Staubli VAL3: gripper.pgx

public program gripper(num nOpen (dimensions=1))
begin
  //nOpen = 0 - close gripper
  //nOpen = 1 - open gripper
  //
  switch nOpen
    case 0
      close(flange)
    break
    case 1
      open(flange)
    break
    default
      logMsg("gripper(): nOpen = "+toString("",nOpen))
    break
  endSwitch
end
